FUNCTION_BLOCK DamperControl
VAR_INPUT
	EN: BOOL;
	Interval: TIME;
	StartTime: TIME_OF_DAY;
	AlarmOnlyOnExercise: bool;
END_VAR
VAR_OUTPUT
	ENO: BOOL;
END_VAR
VAR
END_VAR

ENO := EN;

END_FUNCTION_BLOCK

(* stored: Version 1.1.0.1, ProductVersion 3.1.4024.3
   POU DamperControl: Id {beee9bde-37af-436a-89f9-427fdbc4e4bf}, SpecialFunc None *)
